FUNCTION_BLOCK FB_Cluster_Control
VAR_INPUT
	i_rs_start_auto : ARRAY[1..rs_count] OF BOOL;
	i_rs_stop		: ARRAY[1..rs_count] OF BOOL;
	
END_VAR
VAR_OUTPUT
END_VAR
VAR
	rs_control 			: ARRAY[1..rs_count] OF FB_ReactorSet_Control;
	reactor_set			: ARRAY[1..rs_count] OF FB_ReactorSet;
	rs_error			: BOOL;
	
	utilities_control 	: FB_Utilities_Control;
	
	idx_rs 				: UINT;
	
	{attribute 'to_string'}
	state_cluster		: (Idle := 0, Warmup := 1, Ready := 2, Cycling := 3, Shutdown := 4, Error); 
	
	stop_rs_cmd			: ARRAY[1..rs_count] OF  INT;
	shutdown_util_cmd	: BOOL;
END_VAR

IF hmi.cluster_state_cmd = E_Cluster_State_Cmd.Shutdown AND  state_cluster <> Cycling THEN 
	state_cluster := Shutdown;
END_IF

CASE state_cluster OF 
	
	Idle : 
		utilities_control.i_state_req := E_Cluster_State_Cmd.Idle;
		IF hmi.cluster_state_cmd = E_Cluster_State_Cmd.Warmup THEN 
			state_cluster := Warmup;
		END_IF
		
	Warmup:	
		utilities_control.i_state_req := E_Util_State_Cmd.Warmup;
		IF NOT utilities_control.in_bop_warmup_sts.error  THEN 
			IF utilities_control.in_bop_warmup_sts.completed THEN 
				state_cluster := Ready;
			END_IF
		ELSE
			state_cluster := Error;
		END_IF		
		
	Ready :
		utilities_control.i_state_req := E_Util_State_Cmd.Activate;
		
		IF  NOT utilities_control.o_util_error AND NOT rs_error THEN
			IF  utilities_control.in_bop_activate_sts.completed AND hmi.cluster_state_cmd = E_Cluster_State_Cmd.Cycling THEN 
				state_cluster := Cycling;
			END_IF
		ELSE
			state_cluster := Error;
		END_IF
		
	Cycling :
	
		FOR idx_rs := 1 TO rs_count DO 
			utilities_control.i_cooling_pump_req.rs_number := idx_rs;
			reactor_set[idx_rs]( i_seq_req 				:= rs_control[idx_rs].SeqState_Sts,
								 i_cooling_pump_sts 	:= utilities_control.CoolingPump_Sts,
								 i_deadair_pump_sts 	:= utilities_control.DeadAirPump_Sts,
								 i_steam_system_sts 	:= utilities_control.SteamSystem_Sts,
								 i_purge_assist_sts 	:= utilities_control.PurgeAssist_Sts,
								 o_adsorption_seq_sts 	=> rs_control[idx_rs].i_adsorption_seq_sts,
								 o_airpress_seq_sts		=> rs_control[idx_rs].i_airpress_seq_sts,
								 o_evac_seq_sts 		=> rs_control[idx_rs].i_evac_seq_sts,
								 o_desorption_seq_sts 	=> rs_control[idx_rs].i_desorption_seq_sts,
								 o_cooling_seq_sts		=> rs_control[idx_rs].i_cooling_seq_sts,
								 o_cooling_pump_req		=> utilities_control.i_cooling_pump_req.request_cmd,
								 o_deadair_pump_req		=> utilities_control.i_deadair_pump_req.request_cmd,
								 o_steam_system_req		=> utilities_control.i_steam_system_req.request_cmd,
								 o_purge_assist_req		=> utilities_control.i_purge_assist_req.request_cmd
								);
			
			rs_control[idx_rs]( i_rs_number := idx_rs,
								i_start_cycle := i_rs_start_auto[idx_rs] AND NOT reactor_set[idx_rs].o_error_active,
								//i_stop_cmd := i_rs_stop[idx_rs],
								io_stop_cmd := stop_rs_cmd[idx_rs]
							  );
							  
			
			utilities_control.CoolingPump_Control();
			utilities_control.DeadAirPump_Control();
			
		END_FOR
		
		
		IF  hmi.cluster_state_cmd = E_Cluster_State_Cmd.Shutdown AND Get_All_RS_Done_Sts() THEN 
			state_cluster := Shutdown;
		END_IF
		
	Shutdown : 
		
		utilities_control.i_state_req := E_Util_State_Cmd.Shutdown;
		IF NOT utilities_control.in_bop_shutdown_sts.error THEN 
			IF utilities_control.in_bop_shutdown_sts.completed THEN 
				state_cluster := Idle;
			END_IF
		ELSE
			state_cluster := Error;	
		END_IF
	
	Error : 
		
		IF hmi.cluster_state_cmd = E_Cluster_State_Cmd.Reset_Fault THEN 
			utilities_control.i_state_req := E_Util_State_Cmd.Reset_Fault;
		END_IF
		IF  NOT utilities_control.o_util_error THEN 
				state_cluster := Idle;
		END_IF
		
		
END_CASE

//utilities_control();
utilities_control.State_Machine();

METHOD Get_All_RS_Done_Sts : BOOL
VAR
	rs_done : BOOL;
END_VAR
rs_done := rs_control[1].o_Done;
FOR idx_rs := 2 TO rs_count DO 
	rs_done := rs_done AND rs_control[idx_rs].o_Done;
END_FOR
Get_All_RS_Done_Sts := rs_done;
END_METHOD

END_FUNCTION_BLOCK

(* stored: Version 1.1.0.1, ProductVersion 3.1.4024.12
   POU FB_Cluster_Control: Id {6fd5e4a5-e99d-4b99-9ff7-8b5ec4c922f0}, SpecialFunc None
   Method Get_All_RS_Done_Sts: Id {7304ccc2-7947-447d-8057-95279c90ae71} *)
